// TIA Portal V17 export
// export: Created 2025-03-05T08:01:18.8898414Z, ExportSetting WithDefaults, DisplayName Totally Integrated Automation Portal, DisplayVersion V17 Update 8, DisplayName TIA Portal Openness, DisplayVersion V17 Update 8, DisplayName TIA Portal Version Control Interface, DisplayVersion V17, DisplayName SINAMICS Startdrive Advanced, DisplayVersion V17 SP2, DisplayName SINAMICS Startdrive G110M, G120, G120C, G120D, G120P, G115D, DisplayVersion V17 SP2, DisplayName SINAMICS Startdrive G130, G150, S120, S150, SINAMICS MV, S210, DisplayVersion V17 SP2, DisplayName STEP 7 Professional, DisplayVersion V17 Update 8, DisplayName SINUMERIK ONE STEP 7 Toolbox, DisplayVersion V17 Update 12, DisplayName SINUMERIK 840D sl STEP 7 Toolbox, DisplayVersion V17 Update 12, DisplayName STEP 7 Safety, DisplayVersion V17 Update 6, DisplayName WinCC Advanced, DisplayVersion V17 Update 8
FUNCTION "FC6800_UNIT_02_UP_SEALING_STRUCTURE" : Void   // FC6800, LAD
{ S7_Optimized_Access := 'TRUE' }
VERSION : 0.1
// stored: AutoNumber false, IsIECCheckEnabled false, SetENOAutomatically false, UDAEnableTagReadback false
   VAR_TEMP
      INPUTS_MASK : Byte;   // INPUTS_MASK
      O_BYTE_0 : Struct   // OPTIONS BYTE 0
         CLOSED_INPUT_1 : Bool;   // CLOSED INPUT 1 OPTION
         CLOSED_INPUT_2 : Bool;   // CLOSED INPUT OPTION
         OPEN_INPUT_1 : Bool;   // OPEN INPUT 1 OPTION
         OPEN_INPUT_2 : Bool;   // OPEN INPUT 2 OPTION
         SPARE_4 : Bool;   // SPARE OPTION
         SPARE_5 : Bool;   // SPARE OPTION
         SPARE_6 : Bool;   // SPARE OPTION
         SPARE_7 : Bool;   // SPARE OPTION
      END_STRUCT;
      OPTIONS_0 : Byte;   // OPTIONS 0
      UNIT_ALARM : UInt;
      STATION_ALARM : UInt;
   END_VAR
   VAR CONSTANT
      FC_NUMBER : DInt := 6800;
   END_VAR
   VAR_TEMP   // added for the SCL form of the ladder/FBD networks
      _w1 : Bool;
   END_VAR
BEGIN

REGION Network 1: TEMPORAL (HAY QUE PONER ESTA A 1 PARA PODER ACTIVAR LAS OTRAS VALVULAS)
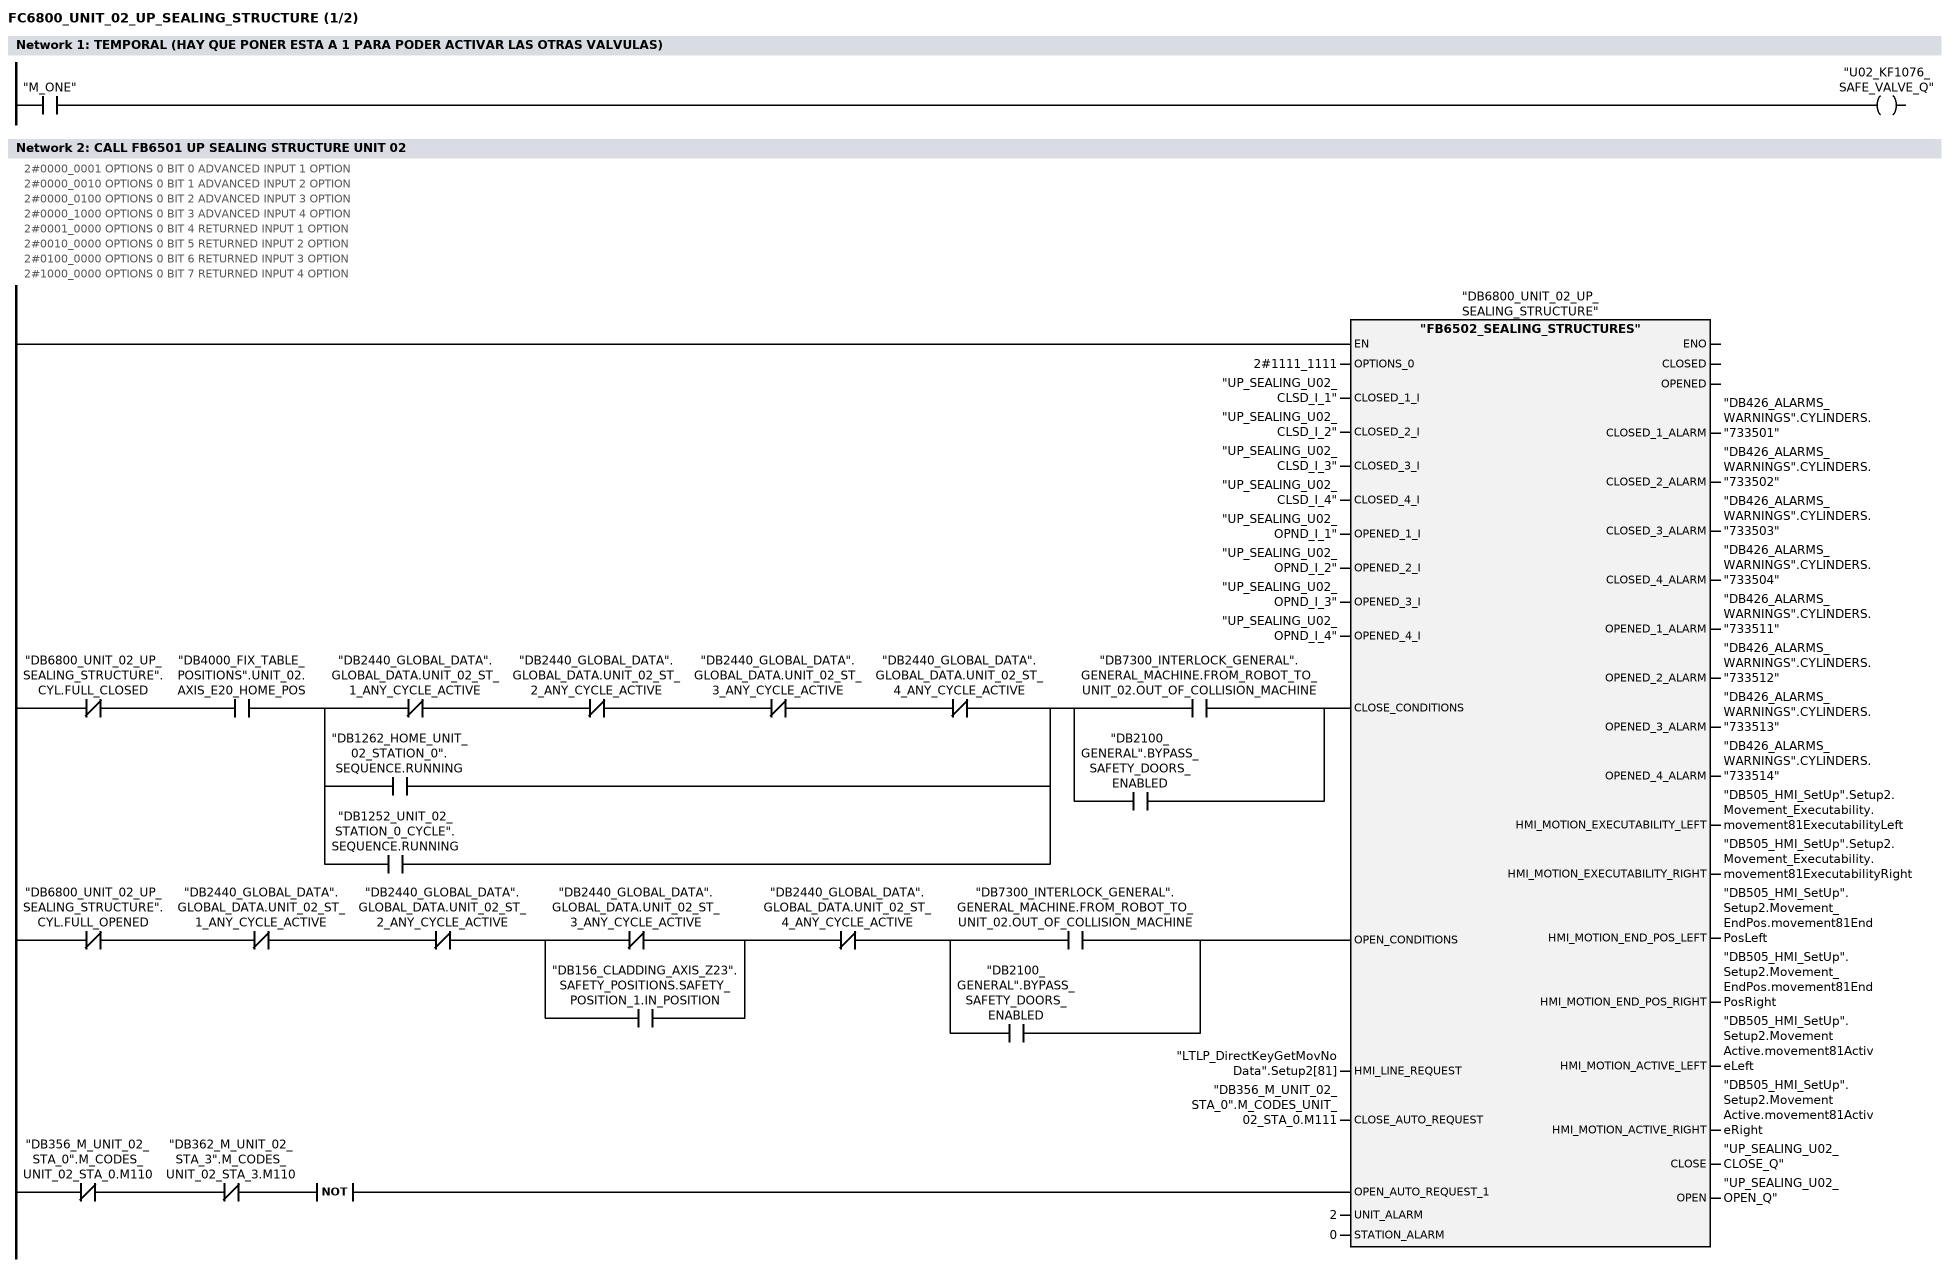
   RUNG wire#powerrail
      Contact( "M_ONE" )
      Coil( "U02_KF1076_SAFE_VALVE_Q" )
   END_RUNG
   // the same network as SCL:
   "U02_KF1076_SAFE_VALVE_Q" := "M_ONE";
END_REGION

REGION Network 2: CALL FB6501 UP SEALING STRUCTURE UNIT 02
   // 2#0000_0001 OPTIONS 0 BIT 0 ADVANCED INPUT 1 OPTION
   // 2#0000_0010 OPTIONS 0 BIT 1 ADVANCED INPUT 2 OPTION
   // 2#0000_0100 OPTIONS 0 BIT 2 ADVANCED INPUT 3 OPTION
   // 2#0000_1000 OPTIONS 0 BIT 3 ADVANCED INPUT 4 OPTION
   // 2#0001_0000 OPTIONS 0 BIT 4 RETURNED INPUT 1 OPTION
   // 2#0010_0000 OPTIONS 0 BIT 5 RETURNED INPUT 2 OPTION
   // 2#0100_0000 OPTIONS 0 BIT 6 RETURNED INPUT 3 OPTION
   // 2#1000_0000 OPTIONS 0 BIT 7 RETURNED INPUT 4 OPTION
   RUNG wire#powerrail
      "DB6800_UNIT_02_UP_SEALING_STRUCTURE"(CLOSE_CONDITIONS := wire#w3, OPEN_CONDITIONS := wire#w7, OPEN_AUTO_REQUEST_1 := wire#w8, OPTIONS_0 := 2#1111_1111, CLOSED_1_I := "UP_SEALING_U02_CLSD_I_1", CLOSED_2_I := "UP_SEALING_U02_CLSD_I_2", CLOSED_3_I := "UP_SEALING_U02_CLSD_I_3", CLOSED_4_I := "UP_SEALING_U02_CLSD_I_4", OPENED_1_I := "UP_SEALING_U02_OPND_I_1", OPENED_2_I := "UP_SEALING_U02_OPND_I_2", OPENED_3_I := "UP_SEALING_U02_OPND_I_3", OPENED_4_I := "UP_SEALING_U02_OPND_I_4", HMI_LINE_REQUEST := "LTLP_DirectKeyGetMovNoData".Setup2[81], CLOSE_AUTO_REQUEST := "DB356_M_UNIT_02_STA_0".M_CODES_UNIT_02_STA_0.M111, UNIT_ALARM := 2, STATION_ALARM := 0, CLOSED =>, OPENED =>, CLOSED_1_ALARM => "DB426_ALARMS_WARNINGS".CYLINDERS."733501", CLOSED_2_ALARM => "DB426_ALARMS_WARNINGS".CYLINDERS."733502", CLOSED_3_ALARM => "DB426_ALARMS_WARNINGS".CYLINDERS."733503", CLOSED_4_ALARM => "DB426_ALARMS_WARNINGS".CYLINDERS."733504", OPENED_1_ALARM => "DB426_ALARMS_WARNINGS".CYLINDERS."733511", OPENED_2_ALARM => "DB426_ALARMS_WARNINGS".CYLINDERS."733512", OPENED_3_ALARM => "DB426_ALARMS_WARNINGS".CYLINDERS."733513", OPENED_4_ALARM => "DB426_ALARMS_WARNINGS".CYLINDERS."733514", HMI_MOTION_EXECUTABILITY_LEFT => "DB505_HMI_SetUp".Setup2.Movement_Executability.movement81ExecutabilityLeft, HMI_MOTION_EXECUTABILITY_RIGHT => "DB505_HMI_SetUp".Setup2.Movement_Executability.movement81ExecutabilityRight, HMI_MOTION_END_POS_LEFT => "DB505_HMI_SetUp".Setup2.Movement_EndPos.movement81EndPosLeft, HMI_MOTION_END_POS_RIGHT => "DB505_HMI_SetUp".Setup2.Movement_EndPos.movement81EndPosRight, HMI_MOTION_ACTIVE_LEFT => "DB505_HMI_SetUp".Setup2.MovementActive.movement81ActiveLeft, HMI_MOTION_ACTIVE_RIGHT => "DB505_HMI_SetUp".Setup2.MovementActive.movement81ActiveRight, CLOSE => "UP_SEALING_U02_CLOSE_Q", OPEN => "UP_SEALING_U02_OPEN_Q")
   END_RUNG
   RUNG wire#powerrail
      I_Contact( "DB6800_UNIT_02_UP_SEALING_STRUCTURE".CYL.FULL_CLOSED )
      Contact( "DB4000_FIX_TABLE_POSITIONS".UNIT_02.AXIS_E20_HOME_POS )
      wire#w1
      I_Contact( "DB2440_GLOBAL_DATA".GLOBAL_DATA.UNIT_02_ST_1_ANY_CYCLE_ACTIVE )
      I_Contact( "DB2440_GLOBAL_DATA".GLOBAL_DATA.UNIT_02_ST_2_ANY_CYCLE_ACTIVE )
      I_Contact( "DB2440_GLOBAL_DATA".GLOBAL_DATA.UNIT_02_ST_3_ANY_CYCLE_ACTIVE )
      I_Contact( "DB2440_GLOBAL_DATA".GLOBAL_DATA.UNIT_02_ST_4_ANY_CYCLE_ACTIVE )
      wire#w2
      Contact( "DB7300_INTERLOCK_GENERAL".GENERAL_MACHINE.FROM_ROBOT_TO_UNIT_02.OUT_OF_COLLISION_MACHINE )
   END_RUNG wire#w3
   RUNG wire#w1
      Contact( "DB1262_HOME_UNIT_02_STATION_0".SEQUENCE.RUNNING )
   END_RUNG wire#w2
   RUNG wire#w1
      Contact( "DB1252_UNIT_02_STATION_0_CYCLE".SEQUENCE.RUNNING )
   END_RUNG wire#w2
   RUNG wire#w2
      Contact( "DB2100_GENERAL".BYPASS_SAFETY_DOORS_ENABLED )
   END_RUNG wire#w3
   RUNG wire#powerrail
      I_Contact( "DB6800_UNIT_02_UP_SEALING_STRUCTURE".CYL.FULL_OPENED )
      I_Contact( "DB2440_GLOBAL_DATA".GLOBAL_DATA.UNIT_02_ST_1_ANY_CYCLE_ACTIVE )
      I_Contact( "DB2440_GLOBAL_DATA".GLOBAL_DATA.UNIT_02_ST_2_ANY_CYCLE_ACTIVE )
      wire#w4
      I_Contact( "DB2440_GLOBAL_DATA".GLOBAL_DATA.UNIT_02_ST_3_ANY_CYCLE_ACTIVE )
      wire#w5
      I_Contact( "DB2440_GLOBAL_DATA".GLOBAL_DATA.UNIT_02_ST_4_ANY_CYCLE_ACTIVE )
      wire#w6
      Contact( "DB7300_INTERLOCK_GENERAL".GENERAL_MACHINE.FROM_ROBOT_TO_UNIT_02.OUT_OF_COLLISION_MACHINE )
   END_RUNG wire#w7
   RUNG wire#w4
      Contact( "DB156_CLADDING_AXIS_Z23".SAFETY_POSITIONS.SAFETY_POSITION_1.IN_POSITION )
   END_RUNG wire#w5
   RUNG wire#w6
      Contact( "DB2100_GENERAL".BYPASS_SAFETY_DOORS_ENABLED )
   END_RUNG wire#w7
   RUNG wire#powerrail
      I_Contact( "DB356_M_UNIT_02_STA_0".M_CODES_UNIT_02_STA_0.M110 )
      I_Contact( "DB362_M_UNIT_02_STA_3".M_CODES_UNIT_02_STA_3.M110 )
      Not()
   END_RUNG wire#w8
   // the same network as SCL:
   "DB6800_UNIT_02_UP_SEALING_STRUCTURE"(OPTIONS_0 := 2#1111_1111,   // "FB6502_SEALING_STRUCTURES"
                           CLOSED_1_I := "UP_SEALING_U02_CLSD_I_1",
                           CLOSED_2_I := "UP_SEALING_U02_CLSD_I_2",
                           CLOSED_3_I := "UP_SEALING_U02_CLSD_I_3",
                           CLOSED_4_I := "UP_SEALING_U02_CLSD_I_4",
                           OPENED_1_I := "UP_SEALING_U02_OPND_I_1",
                           OPENED_2_I := "UP_SEALING_U02_OPND_I_2",
                           OPENED_3_I := "UP_SEALING_U02_OPND_I_3",
                           OPENED_4_I := "UP_SEALING_U02_OPND_I_4",
                           CLOSE_CONDITIONS := NOT "DB6800_UNIT_02_UP_SEALING_STRUCTURE".CYL.FULL_CLOSED AND "DB4000_FIX_TABLE_POSITIONS".UNIT_02.AXIS_E20_HOME_POS AND ((NOT "DB2440_GLOBAL_DATA".GLOBAL_DATA.UNIT_02_ST_1_ANY_CYCLE_ACTIVE AND NOT "DB2440_GLOBAL_DATA".GLOBAL_DATA.UNIT_02_ST_2_ANY_CYCLE_ACTIVE AND NOT "DB2440_GLOBAL_DATA".GLOBAL_DATA.UNIT_02_ST_3_ANY_CYCLE_ACTIVE AND NOT "DB2440_GLOBAL_DATA".GLOBAL_DATA.UNIT_02_ST_4_ANY_CYCLE_ACTIVE) OR "DB1262_HOME_UNIT_02_STATION_0".SEQUENCE.RUNNING OR "DB1252_UNIT_02_STATION_0_CYCLE".SEQUENCE.RUNNING) AND ("DB7300_INTERLOCK_GENERAL".GENERAL_MACHINE.FROM_ROBOT_TO_UNIT_02.OUT_OF_COLLISION_MACHINE OR "DB2100_GENERAL".BYPASS_SAFETY_DOORS_ENABLED),
                           OPEN_CONDITIONS := NOT "DB6800_UNIT_02_UP_SEALING_STRUCTURE".CYL.FULL_OPENED AND NOT "DB2440_GLOBAL_DATA".GLOBAL_DATA.UNIT_02_ST_1_ANY_CYCLE_ACTIVE AND NOT "DB2440_GLOBAL_DATA".GLOBAL_DATA.UNIT_02_ST_2_ANY_CYCLE_ACTIVE AND (NOT "DB2440_GLOBAL_DATA".GLOBAL_DATA.UNIT_02_ST_3_ANY_CYCLE_ACTIVE OR "DB156_CLADDING_AXIS_Z23".SAFETY_POSITIONS.SAFETY_POSITION_1.IN_POSITION) AND NOT "DB2440_GLOBAL_DATA".GLOBAL_DATA.UNIT_02_ST_4_ANY_CYCLE_ACTIVE AND ("DB7300_INTERLOCK_GENERAL".GENERAL_MACHINE.FROM_ROBOT_TO_UNIT_02.OUT_OF_COLLISION_MACHINE OR "DB2100_GENERAL".BYPASS_SAFETY_DOORS_ENABLED),
                           HMI_LINE_REQUEST := "LTLP_DirectKeyGetMovNoData".Setup2[81],
                           CLOSE_AUTO_REQUEST := "DB356_M_UNIT_02_STA_0".M_CODES_UNIT_02_STA_0.M111,
                           OPEN_AUTO_REQUEST_1 := NOT (NOT "DB356_M_UNIT_02_STA_0".M_CODES_UNIT_02_STA_0.M110 AND NOT "DB362_M_UNIT_02_STA_3".M_CODES_UNIT_02_STA_3.M110),
                           UNIT_ALARM := 2,
                           STATION_ALARM := 0,
                           CLOSED_1_ALARM => "DB426_ALARMS_WARNINGS".CYLINDERS."733501",
                           CLOSED_2_ALARM => "DB426_ALARMS_WARNINGS".CYLINDERS."733502",
                           CLOSED_3_ALARM => "DB426_ALARMS_WARNINGS".CYLINDERS."733503",
                           CLOSED_4_ALARM => "DB426_ALARMS_WARNINGS".CYLINDERS."733504",
                           OPENED_1_ALARM => "DB426_ALARMS_WARNINGS".CYLINDERS."733511",
                           OPENED_2_ALARM => "DB426_ALARMS_WARNINGS".CYLINDERS."733512",
                           OPENED_3_ALARM => "DB426_ALARMS_WARNINGS".CYLINDERS."733513",
                           OPENED_4_ALARM => "DB426_ALARMS_WARNINGS".CYLINDERS."733514",
                           HMI_MOTION_EXECUTABILITY_LEFT => "DB505_HMI_SetUp".Setup2.Movement_Executability.movement81ExecutabilityLeft,
                           HMI_MOTION_EXECUTABILITY_RIGHT => "DB505_HMI_SetUp".Setup2.Movement_Executability.movement81ExecutabilityRight,
                           HMI_MOTION_END_POS_LEFT => "DB505_HMI_SetUp".Setup2.Movement_EndPos.movement81EndPosLeft,
                           HMI_MOTION_END_POS_RIGHT => "DB505_HMI_SetUp".Setup2.Movement_EndPos.movement81EndPosRight,
                           HMI_MOTION_ACTIVE_LEFT => "DB505_HMI_SetUp".Setup2.MovementActive.movement81ActiveLeft,
                           HMI_MOTION_ACTIVE_RIGHT => "DB505_HMI_SetUp".Setup2.MovementActive.movement81ActiveRight,
                           CLOSE => "UP_SEALING_U02_CLOSE_Q",
                           OPEN => "UP_SEALING_U02_OPEN_Q");
END_REGION

REGION Network 3: OPERATOR HELP
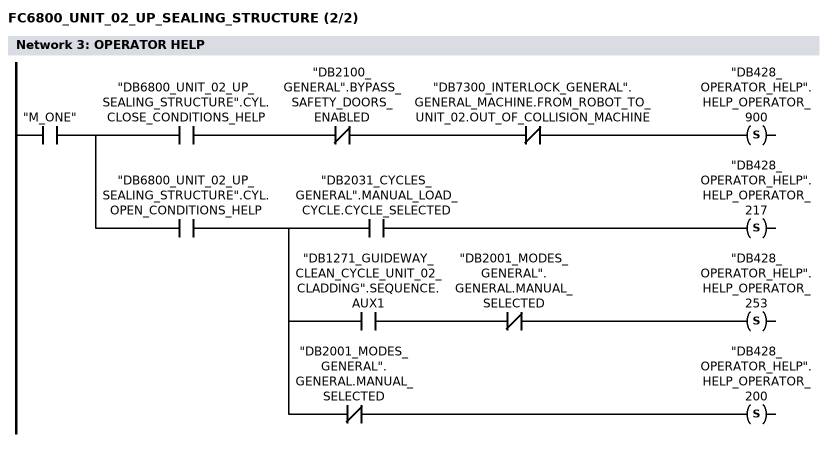
   RUNG wire#powerrail
      Contact( "M_ONE" )
      wire#w1
      Contact( "DB6800_UNIT_02_UP_SEALING_STRUCTURE".CYL.CLOSE_CONDITIONS_HELP )
      I_Contact( "DB2100_GENERAL".BYPASS_SAFETY_DOORS_ENABLED )
      I_Contact( "DB7300_INTERLOCK_GENERAL".GENERAL_MACHINE.FROM_ROBOT_TO_UNIT_02.OUT_OF_COLLISION_MACHINE )
      S_Coil( "DB428_OPERATOR_HELP".HELP_OPERATOR_900 )
   END_RUNG
   RUNG wire#w1
      Contact( "DB6800_UNIT_02_UP_SEALING_STRUCTURE".CYL.OPEN_CONDITIONS_HELP )
      wire#w2
      Contact( "DB2031_CYCLES_GENERAL".MANUAL_LOAD_CYCLE.CYCLE_SELECTED )
      S_Coil( "DB428_OPERATOR_HELP".HELP_OPERATOR_217 )
   END_RUNG
   RUNG wire#w2
      Contact( "DB1271_GUIDEWAY_CLEAN_CYCLE_UNIT_02_CLADDING".SEQUENCE.AUX1 )
      I_Contact( "DB2001_MODES_GENERAL".GENERAL.MANUAL_SELECTED )
      S_Coil( "DB428_OPERATOR_HELP".HELP_OPERATOR_253 )
   END_RUNG
   RUNG wire#w2
      I_Contact( "DB2001_MODES_GENERAL".GENERAL.MANUAL_SELECTED )
      S_Coil( "DB428_OPERATOR_HELP".HELP_OPERATOR_200 )
   END_RUNG
   // the same network as SCL:
   IF "M_ONE" AND "DB6800_UNIT_02_UP_SEALING_STRUCTURE".CYL.CLOSE_CONDITIONS_HELP AND NOT "DB2100_GENERAL".BYPASS_SAFETY_DOORS_ENABLED AND NOT "DB7300_INTERLOCK_GENERAL".GENERAL_MACHINE.FROM_ROBOT_TO_UNIT_02.OUT_OF_COLLISION_MACHINE THEN
       "DB428_OPERATOR_HELP".HELP_OPERATOR_900 := TRUE;
   END_IF;
   #_w1 := "M_ONE" AND "DB6800_UNIT_02_UP_SEALING_STRUCTURE".CYL.OPEN_CONDITIONS_HELP;
   IF #_w1 AND "DB2031_CYCLES_GENERAL".MANUAL_LOAD_CYCLE.CYCLE_SELECTED THEN
       "DB428_OPERATOR_HELP".HELP_OPERATOR_217 := TRUE;
   END_IF;
   IF #_w1 AND "DB1271_GUIDEWAY_CLEAN_CYCLE_UNIT_02_CLADDING".SEQUENCE.AUX1 AND NOT "DB2001_MODES_GENERAL".GENERAL.MANUAL_SELECTED THEN
       "DB428_OPERATOR_HELP".HELP_OPERATOR_253 := TRUE;
   END_IF;
   IF #_w1 AND NOT "DB2001_MODES_GENERAL".GENERAL.MANUAL_SELECTED THEN
       "DB428_OPERATOR_HELP".HELP_OPERATOR_200 := TRUE;
   END_IF;
END_REGION
END_FUNCTION
